(* CoDeSys 2.3 export: ST_SERIAL64BYTEOUT.EXP *)

(* Data type *)
TYPE ST_Serial64ByteOut :
STRUCT
	wControl:WORD;
	aData   :ARRAY[0..63] OF BYTE;
END_STRUCT
END_TYPE
